// TIA Portal V16 export
// export: Created 2022-11-17T15:49:45.2202364Z, ExportSetting WithDefaults, DisplayName Totally Integrated Automation Portal, DisplayVersion V16 Update 6, DisplayName TIA Portal Version Control Interface, DisplayVersion V16 Update 2, DisplayName TIA Portal Openness, DisplayVersion V16 Update 6, DisplayName SINAMICS Startdrive Advanced, DisplayVersion V16 Update 5, DisplayName SINAMICS Startdrive G130, G150, S120, S150, SINAMICS MV, S210, DisplayVersion V16 Update 5, DisplayName SINAMICS Startdrive G110M, G120, G120C, G120D, G120P, G115D, DisplayVersion V16 Update 5, DisplayName STEP 7 Professional, DisplayVersion V16 Update 6, DisplayName STEP 7 Safety, DisplayVersion V16, DisplayName WinCC Advanced, DisplayVersion V16 Update 6
DATA_BLOCK "DB244_Program6"   // DB244
{ S7_Optimized_Access := 'FALSE' }
AUTHOR : Robopac
VERSION : 0.0
// stored: AutoNumber false, IsOnlyStoredInLoadMemory false, IsWriteProtectedInAS false
   VAR RETAIN
      Program6 { S7_SetPoint := 'True'} : "DatiProgramma";
   END_VAR
BEGIN
   Program6.Wrapping := TRUE;
   Program6.TopLenght := 500;
   Program6.TopRelease := 0;
   Program6.TopDown := 0;
   Program6.Top := 4;
   Program6.PressurePTime := 0;
   Program6.LifterTime := 0;
   Program6.RevOverContrast := 1;
   Program6.RopeEndCycle := 16#02;
   Program6.Spare4 := 16#01;
   Program6.RopeTime := 1500;
   Program6.RevOverClamp := 1;
   Program6.FilmForceFinalRev := 10;
   Program6.FilmPrestretchFinalRev := 100;
   Program6.ArmSpeed := 100;
   Program6.CarriageDown4Top := 500;
   Program6.TopDownTime := 1500;
   Program6.LapsUnderTop := 0;
   Program6.Spare6 := 0;
   Program6.Spare7 := 0;
   Program6.Spare8 := 0;
   Program6.Spare9 := 0;
   Program6.Spare10 := 0;
   Program6.Spare11 := 0;
   Program6.Spare12 := 0;
   Program6.Overlap0_1 := 0;
   Program6.Height1 := 130;
   Program6.Landmark1 := FALSE;
   Program6.Lifter1 := FALSE;
   Program6.SpareBit1H1 := FALSE;
   Program6.Airblower1 := TRUE;
   Program6.NextStep1 := TRUE;
   Program6.PressureP1 := TRUE;
   Program6.SpareByte2H1 := 16#00;
   Program6.Revolution1 := 1;
   Program6.RopeUnit1_1 := 16#01;
   Program6.RopeUnit1_2 := 16#01;
   Program6.FilmForce1 := 5;
   Program6.FilmPrestretch1 := 200;
   Program6.Spare3H1 := 0;
   Program6.Spare49 := 0;
   Program6.Spare50 := 0;
   Program6.Spare51 := 0;
   Program6.Spare52 := 0;
   Program6.Spare53 := 0;
   Program6.Overlap1_2 := 0;
   Program6.Height2 := 50;
   Program6.Landmark2 := FALSE;
   Program6.Lifter2 := FALSE;
   Program6.SpareBit1H2 := FALSE;
   Program6.Airblower2 := TRUE;
   Program6.NextStep2 := TRUE;
   Program6.PressureP2 := TRUE;
   Program6.SpareByte2H2 := 16#00;
   Program6.Revolution2 := 1;
   Program6.RopeUnit2_1 := 16#01;
   Program6.RopeUnit2_2 := 16#01;
   Program6.FilmForce2 := 20;
   Program6.FilmPrestretch2 := 200;
   Program6.Spare3H2 := 0;
   Program6.Spare54 := 0;
   Program6.Spare55 := 0;
   Program6.Spare56 := 0;
   Program6.Spare57 := 0;
   Program6.Spare58 := 0;
   Program6.Overlap2_3 := 100;
   Program6.Height3 := -50;
   Program6.Landmark3 := TRUE;
   Program6.Lifter3 := FALSE;
   Program6.SpareBit1H3 := FALSE;
   Program6.Airblower3 := TRUE;
   Program6.NextStep3 := TRUE;
   Program6.PressureP3 := TRUE;
   Program6.SpareByte2H3 := 16#00;
   Program6.Revolution3 := 2;
   Program6.RopeUnit3_1 := 16#01;
   Program6.RopeUnit3_2 := 16#01;
   Program6.FilmForce3 := 30;
   Program6.FilmPrestretch3 := 200;
   Program6.Spare3H3 := 0;
   Program6.Spare59 := 0;
   Program6.Spare60 := 0;
   Program6.Spare61 := 380;
   Program6.Spare62 := 2800;
   Program6.Spare63 := 0;
   Program6.Overlap3_4 := 100;
   Program6.Height4 := 100;
   Program6.Landmark4 := FALSE;
   Program6.Lifter4 := FALSE;
   Program6.SpareBit1H4 := FALSE;
   Program6.Airblower4 := TRUE;
   Program6.NextStep4 := TRUE;
   Program6.PressureP4 := TRUE;
   Program6.SpareByte2H4 := 16#00;
   Program6.Revolution4 := 3;
   Program6.RopeUnit4_1 := 16#02;
   Program6.RopeUnit4_2 := 16#02;
   Program6.FilmForce4 := 30;
   Program6.FilmPrestretch4 := 200;
   Program6.Spare3H4 := 0;
   Program6.Spare64 := 0;
   Program6.Spare65 := 0;
   Program6.Spare66 := 0;
   Program6.Spare67 := 0;
   Program6.Spare68 := 0;
   Program6.Overlap4_5 := 0;
   Program6.Height5 := 50;
   Program6.Landmark5 := FALSE;
   Program6.Lifter5 := FALSE;
   Program6.SpareBit1H5 := FALSE;
   Program6.Airblower5 := TRUE;
   Program6.NextStep5 := FALSE;
   Program6.PressureP5 := FALSE;
   Program6.SpareByte2H5 := 16#00;
   Program6.Revolution5 := 1;
   Program6.RopeUnit5_1 := 16#01;
   Program6.RopeUnit5_2 := 16#01;
   Program6.FilmForce5 := 30;
   Program6.FilmPrestretch5 := 200;
   Program6.Spare3H5 := 0;
   Program6.Spare69 := 0;
   Program6.Spare70 := 0;
   Program6.Spare71 := 0;
   Program6.Spare72 := 0;
   Program6.Spare73 := 0;
   Program6.Overlap5_6 := 100;
   Program6.Height6 := 50;
   Program6.Landmark6 := FALSE;
   Program6.Lifter6 := FALSE;
   Program6.SpareBit1H6 := FALSE;
   Program6.Airblower6 := TRUE;
   Program6.NextStep6 := FALSE;
   Program6.PressureP6 := FALSE;
   Program6.SpareByte2H6 := 16#00;
   Program6.Revolution6 := 2;
   Program6.RopeUnit6_1 := 16#02;
   Program6.RopeUnit6_2 := 16#01;
   Program6.FilmForce6 := 20;
   Program6.FilmPrestretch6 := 200;
   Program6.Spare3H6 := 0;
   Program6.Spare74 := 0;
   Program6.Spare75 := 0;
   Program6.Spare76 := 0;
   Program6.Spare77 := 0;
   Program6.Spare78 := 0;
   Program6.Overlap6_7 := 0;
   Program6.Height7 := 0;
   Program6.Landmark7 := FALSE;
   Program6.Lifter7 := FALSE;
   Program6.SpareBit1H7 := FALSE;
   Program6.Airblower7 := FALSE;
   Program6.NextStep7 := TRUE;
   Program6.PressureP7 := FALSE;
   Program6.SpareByte2H7 := 16#00;
   Program6.Revolution7 := 1;
   Program6.RopeUnit7_1 := 16#01;
   Program6.RopeUnit7_2 := 16#01;
   Program6.FilmForce7 := 0;
   Program6.FilmPrestretch7 := 100;
   Program6.Spare3H7 := 0;
   Program6.Spare79 := 0;
   Program6.Spare80 := 0;
   Program6.Spare81 := 0;
   Program6.Spare82 := 0;
   Program6.Spare83 := 0;
   Program6.Overlap7_8 := 0;
   Program6.Height8 := 0;
   Program6.Landmark8 := FALSE;
   Program6.Lifter8 := FALSE;
   Program6.SpareBit1H8 := FALSE;
   Program6.Airblower8 := FALSE;
   Program6.NextStep8 := TRUE;
   Program6.PressureP8 := FALSE;
   Program6.SpareByte2H8 := 16#00;
   Program6.Revolution8 := 1;
   Program6.RopeUnit8_1 := 16#01;
   Program6.RopeUnit8_2 := 16#01;
   Program6.FilmForce8 := 0;
   Program6.FilmPrestretch8 := 100;
   Program6.Spare3H8 := 0;
   Program6.Spare84 := 0;
   Program6.Spare85 := 0;
   Program6.Spare86 := 0;
   Program6.Spare87 := 0;
   Program6.Spare88 := 0;
   Program6.Overlap8_9 := 0;
   Program6.Height9 := 0;
   Program6.Landmark9 := FALSE;
   Program6.Lifter9 := FALSE;
   Program6.SpareBit1H9 := FALSE;
   Program6.Airblower9 := FALSE;
   Program6.NextStep9 := TRUE;
   Program6.PressureP9 := FALSE;
   Program6.SpareByte2H9 := 16#00;
   Program6.Revolution9 := 1;
   Program6.RopeUnit9_1 := 16#01;
   Program6.RopeUnit9_2 := 16#01;
   Program6.FilmForce9 := 0;
   Program6.FilmPrestretch9 := 100;
   Program6.Spare3H9 := 0;
   Program6.Spare89 := 0;
   Program6.Spare90 := 0;
   Program6.Spare91 := 0;
   Program6.Spare92 := 0;
   Program6.Spare93 := 0;
   Program6.Overlap9_10 := 0;
   Program6.Height10 := 0;
   Program6.Landmark10 := FALSE;
   Program6.Lifter10 := FALSE;
   Program6.SpareBit1H10 := FALSE;
   Program6.Airblower10 := FALSE;
   Program6.NextStep10 := FALSE;
   Program6.PressureP10 := FALSE;
   Program6.SpareByte2H10 := 16#00;
   Program6.Revolution10 := 1;
   Program6.RopeUnit10_1 := 16#01;
   Program6.RopeUnit10_2 := 16#01;
   Program6.FilmForce10 := 0;
   Program6.FilmPrestretch10 := 100;
   Program6.Spare3H10 := 0;
   Program6.Spare94 := 0;
   Program6.Spare95 := 0;
   Program6.Spare96 := 0;
   Program6.Spare97 := 0;
   Program6.Spare98 := 0;
   Program6.Overlap10_11 := 0;
   Program6.Height11 := 0;
   Program6.Landmark11 := FALSE;
   Program6.Lifter11 := FALSE;
   Program6.SpareBit1H11 := FALSE;
   Program6.Airblower11 := FALSE;
   Program6.NextStep11 := TRUE;
   Program6.PressureP11 := FALSE;
   Program6.SpareByte2H11 := 16#00;
   Program6.Revolution11 := 1;
   Program6.RopeUnit11_1 := 16#01;
   Program6.RopeUnit11_2 := 16#01;
   Program6.FilmForce11 := 0;
   Program6.FilmPrestretch11 := 100;
   Program6.Spare3H11 := 0;
   Program6.Spare99 := 0;
   Program6.Spare100 := 0;
   Program6.Spare101 := 0;
   Program6.Spare102 := 0;
   Program6.Spare103 := 0;
   Program6.Overlap11_12 := 0;
   Program6.Height12 := 0;
   Program6.Landmark12 := FALSE;
   Program6.Lifter12 := FALSE;
   Program6.SpareBit1H12 := FALSE;
   Program6.Airblower12 := FALSE;
   Program6.NextStep12 := FALSE;
   Program6.PressureP12 := FALSE;
   Program6.SpareByte2H12 := 16#00;
   Program6.Revolution12 := 1;
   Program6.RopeUnit12_1 := 16#01;
   Program6.RopeUnit12_2 := 16#01;
   Program6.FilmForce12 := 0;
   Program6.FilmPrestretch12 := 100;
   Program6.Spare3H12 := 0;
   Program6.Spare104 := 0;
   Program6.Spare105 := 0;
   Program6.Spare106 := 0;
   Program6.Spare107 := 0;
   Program6.Spare108 := 0;
END_DATA_BLOCK
